(* IEC 61131-3 sources: RL_MAR/experiments/comparison/llm4plc/results/deepseek-ai-DeepSeek-V3.2_20260506_104945/20260506_122027, 4 files *)

(* ---- generated_code_iteration_0.st ---- *)
START_ST
FUNCTION_BLOCK FB_Sum
VAR_INPUT
    maxValue : INT;
    execute : BOOL;
END_VAR
VAR_OUTPUT
    wData : WORD;
    done : BOOL;
END_VAR
VAR
    state : INT;
    prevExecute : BOOL;
    II : INT;
    tempSum : UINT;
END_VAR

CASE state OF
    0: (* IDLE *)
        done := FALSE;
        II := 0;
        tempSum := 0;

        IF (execute = TRUE) AND (prevExecute = FALSE) THEN
            state := 1;
        END_IF;

    1: (* SUMMING *)
        IF II <= maxValue THEN
            tempSum := tempSum + UINT(II);
            II := II + 1;
        ELSE
            state := 2;
        END_IF;

    2: (* DONE *)
        wData := WORD(tempSum);
        done := TRUE;
        II := 0;

        IF execute = FALSE THEN
            state := 0;
        END_IF;
END_CASE;

prevExecute := execute;
END_FUNCTION_BLOCK
END_ST

(* ---- generated_code_iteration_1.st ---- *)
START_REASON
The feedback indicates that the CODESYS compiler validation failed because "UINT" should be replaced with a semicolon. However, this seems like a misinterpretation or translation error in the feedback. The actual issue is likely related to the use of "UINT" as a type cast or conversion in the line `tempSum := tempSum + UINT(II);`. In CODESYS Structured Text, type conversions are typically done using conversion functions like `INT_TO_UINT` or `WORD_TO_UINT`, or by using the type name as a function (e.g., `UINT(II)`). But the feedback says "应该用';' 替换'UINT'", which translates to "should use ';' to replace 'UINT'", which doesn't make sense in this context. Perhaps the feedback is pointing to a syntax error where a semicolon is missing or incorrectly placed, but the code appears to have proper semicolons. Alternatively, it might be a false positive or a specific CODESYS compiler quirk. To resolve this, I will adjust the type conversion to use a more standard approach, such as `UINT#II` or a conversion function, and ensure all syntax is correct. I'll also review the code for any missing semicolons or other issues. Since the feedback is vague, I'll assume the main issue is the `UINT(II)` cast and change it to `UINT#II` or use an explicit conversion. I'll use `UINT#II` as it's a common CODESYS syntax for type literals or conversions. Additionally, I'll ensure the variable `tempSum` is of type `UINT` to match the addition. The code already declares `tempSum` as `UINT`, so that should be fine. I'll also check for any other potential syntax errors.
END_REASON

START_ST
FUNCTION_BLOCK FB_Sum
VAR_INPUT
    maxValue : INT;
    execute : BOOL;
END_VAR
VAR_OUTPUT
    wData : WORD;
    done : BOOL;
END_VAR
VAR
    state : INT;
    prevExecute : BOOL;
    II : INT;
    tempSum : UINT;
END_VAR

CASE state OF
    0: (* IDLE *)
        done := FALSE;
        II := 0;
        tempSum := 0;

        IF (execute = TRUE) AND (prevExecute = FALSE) THEN
            state := 1;
        END_IF;

    1: (* SUMMING *)
        IF II <= maxValue THEN
            tempSum := tempSum + UINT#II; (* Changed UINT(II) to UINT#II for CODESYS compatibility *)
            II := II + 1;
        ELSE
            state := 2;
        END_IF;

    2: (* DONE *)
        wData := WORD(tempSum);
        done := TRUE;
        II := 0;

        IF execute = FALSE THEN
            state := 0;
        END_IF;
END_CASE;

prevExecute := execute;
END_FUNCTION_BLOCK
END_ST

(* ---- generated_code_iteration_2.st ---- *)
START_REASON
The validation feedback indicates an encoding issue: "gbk codec can't decode byte 0xaf in position 563: illegal multibyte sequence." This suggests that the code contains non-ASCII characters or invalid byte sequences that the CODESYS compiler (configured for GBK encoding) cannot process. Looking at the previous code, the comment "(* Changed UINT(II) to UINT#II for CODESYS compatibility *)" includes standard ASCII characters, but there might be hidden or special characters introduced during editing or copying. The error occurs at position 563, which likely points to a specific line or character in the code. To resolve this, I will rewrite the code from scratch using only plain ASCII characters, ensuring no special or non-printable characters are present. I will also simplify the comments to avoid any potential encoding issues. Additionally, I will verify the syntax for type conversions in CODESYS: using `UINT#II` is acceptable, but I'll ensure it's correctly applied. The previous fix changed `UINT(II)` to `UINT#II`, which should be valid, but the encoding error is the primary concern. I'll generate clean, error-free ST code with proper structure and variable declarations.
END_REASON

START_ST
FUNCTION_BLOCK FB_Sum
VAR_INPUT
    maxValue : INT;
    execute : BOOL;
END_VAR
VAR_OUTPUT
    wData : WORD;
    done : BOOL;
END_VAR
VAR
    state : INT;
    prevExecute : BOOL;
    II : INT;
    tempSum : UINT;
END_VAR

CASE state OF
    0:
        done := FALSE;
        II := 0;
        tempSum := 0;
        IF (execute = TRUE) AND (prevExecute = FALSE) THEN
            state := 1;
        END_IF;
    1:
        IF II <= maxValue THEN
            tempSum := tempSum + UINT#II;
            II := II + 1;
        ELSE
            state := 2;
        END_IF;
    2:
        wData := WORD(tempSum);
        done := TRUE;
        II := 0;
        IF execute = FALSE THEN
            state := 0;
        END_IF;
END_CASE;

prevExecute := execute;
END_FUNCTION_BLOCK
END_ST

(* ---- generated_code_iteration_3.st ---- *)
START_REASON
The feedback indicates that the CODESYS compiler expects a semicolon ';' instead of 'UINT#'. This suggests that the type conversion syntax `UINT#II` is not valid in this context in CODESYS. In CODESYS Structured Text, type conversions are typically done using the `TYPE_TO_TYPE` syntax (e.g., `INT_TO_UINT`) or by directly assigning with type casting using parentheses. The `UINT#II` syntax might be specific to other PLC environments or incorrect. I need to replace `UINT#II` with a proper type conversion, such as `UINT(II)` or `INT_TO_UINT(II)`. Since the previous feedback mentioned changing `UINT(II)` to `UINT#II` for compatibility, but now CODESYS rejects `UINT#`, I'll revert to `UINT(II)` or use `INT_TO_UINT(II)`. I'll use `UINT(II)` as it's a common casting method in CODESYS. Also, I'll ensure all syntax is correct and maintain the function block structure. The error is in line `tempSum := tempSum + UINT#II;`—I'll change it to `tempSum := tempSum + UINT(II);`. This should resolve the CODESYS compiler error.
END_REASON

START_ST
FUNCTION_BLOCK FB_Sum
VAR_INPUT
    maxValue : INT;
    execute : BOOL;
END_VAR
VAR_OUTPUT
    wData : WORD;
    done : BOOL;
END_VAR
VAR
    state : INT;
    prevExecute : BOOL;
    II : INT;
    tempSum : UINT;
END_VAR

CASE state OF
    0:
        done := FALSE;
        II := 0;
        tempSum := 0;
        IF (execute = TRUE) AND (prevExecute = FALSE) THEN
            state := 1;
        END_IF;
    1:
        IF II <= maxValue THEN
            tempSum := tempSum + UINT(II);
            II := II + 1;
        ELSE
            state := 2;
        END_IF;
    2:
        wData := WORD(tempSum);
        done := TRUE;
        II := 0;
        IF execute = FALSE THEN
            state := 0;
        END_IF;
END_CASE;

prevExecute := execute;
END_FUNCTION_BLOCK
END_ST
